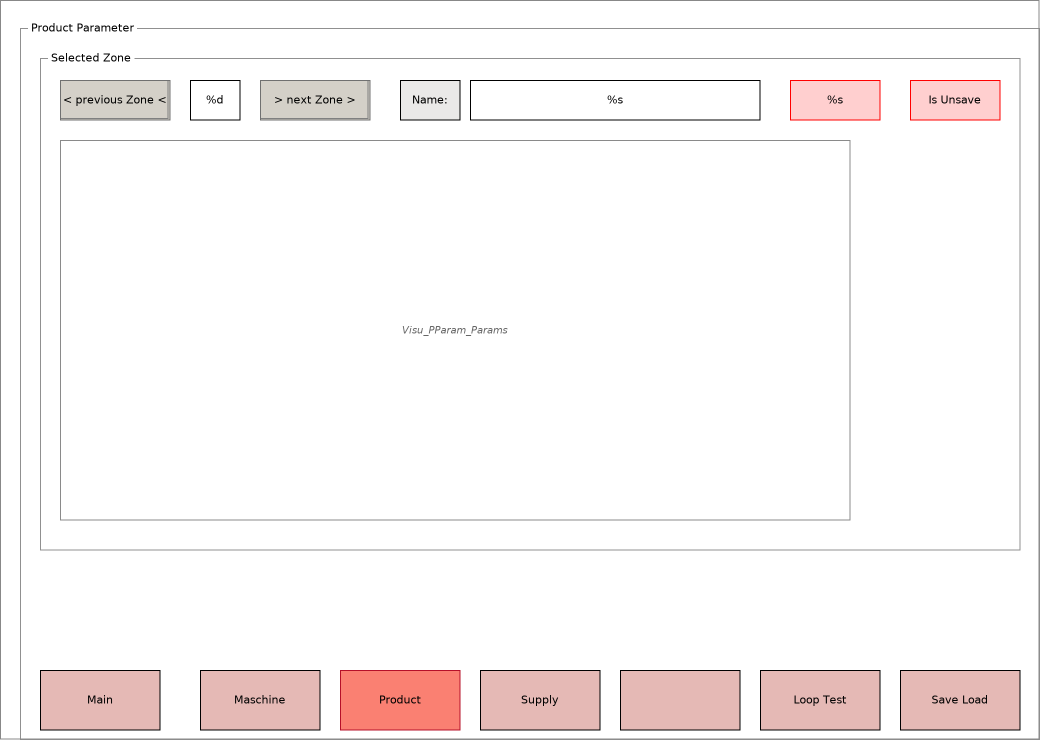
VISUALIZATION Visu_PParam  // 1040x740
    GroupBox (20,20 1020x720), "Product Parameter"
        Rectangle (20,650 120x60), "Main"
            OnMouseClick: change screen: Visu_Main
        Rectangle (880,650 120x60), "Save Load"
            OnMouseClick: change screen: Visu_SaveLoad
        Rectangle (320,650 120x60), "Product"
            OnMouseClick: change screen: Visu_PParam
        GroupBox (20,30 980x500), "Selected Zone"
            Rectangle (150,30 50x40), "%d", text variable: nVisuCount
            Button (20,30 110x40), "< previous Zone <"
                tap bVisuBefore
            Button (220,30 110x40), "> next Zone >"
                tap bVisuNext
            Rectangle (430,30 290x40), "%s", text variable: aaaPfwTempMparamFromHmi[nVisuCount].ZoneName
            Rectangle (360,30 60x40), "Name:"
            Frame (20,90 790x380)
                shows Visu_PParam_Params()
                shows Visu_MParam_ENUM()
                shows Visu_MParam_BOOL()
                shows Visu_MParam_INT()
            Rectangle (870,30 90x40), "Is Unsave", invisible if: Not stParamsUnsave.pParams[nVisuCount]
                OnMouseClick: execute { aaaPfwTempPparamFromHmi[nVisuCount].SaveDelay:=1000; stParamsUnsave.pParams[nVisuCount]:=FALSE; }
        Rectangle (180,650 120x60), "Maschine"
            OnMouseClick: change screen: Visu_MParam
    Rectangle (480,670 120x60), "Supply"
        OnMouseClick: change screen: Visu_Supply
    Rectangle (620,670 120x60)
    Rectangle (760,670 120x60), "Loop Test"
        OnMouseClick: change screen: Visu_LoopTest
    Rectangle (790,80 90x40), "%s", text variable: stMParam_Visu.sInUse, colour toggle: aaaPfwTempMparamFromHmi[nVisuCount].InUse
        OnMouseClick: toggle aaaPfwTempMparamFromHmi[nVisuCount].InUse
        OnMouseClick: execute { stParamsUnsave.mParams[nVisuCount]:=TRUE; }
END_VISUALIZATION

(* stored: Version 1.1.0.1
   Visu Visu_PParam: Id {eff25338-80ea-415c-81d6-5b549848aea3} *)
